INTERFACE I_CommandSteps

METHOD AssemblyEnd : BOOL
VAR_INPUT
END_VAR
END_METHOD

METHOD AssemblyStart : BOOL
VAR_INPUT
END_VAR
END_METHOD

METHOD Board : BOOL
VAR_INPUT
END_VAR
END_METHOD

METHOD BoardInfo : BOOL
VAR_INPUT
END_VAR
END_METHOD

METHOD NailPlate : BOOL
VAR_INPUT
END_VAR
END_METHOD

METHOD TrussInfo : BOOL
VAR_INPUT
END_VAR
END_METHOD

END_INTERFACE

(* stored: Version 1.1.0.1
   Itf I_CommandSteps: Id {5622a179-9d41-4cb7-962d-06a33dfb98f2}
   Method AssemblyEnd: Id {818ab77b-962e-4fb6-a5e7-6dcec8bbe4c1}
   Method AssemblyStart: Id {94786fe6-5b20-4fdd-99b8-7b11813b4a9e}
   Method Board: Id {f1243003-10cd-4ba2-a5df-6c1c4d634ea1}
   Method BoardInfo: Id {5ee4d879-62a4-4eae-8b99-5e765a3268b7}
   Method NailPlate: Id {db76b8a1-b606-4e25-81e5-ec9f253e8fbf}
   Method TrussInfo: Id {90fdfe7b-fd9c-4f05-9a01-d32a876139eb} *)
